// TwinCAT 3 PLC project HARTL_PowerLink_v2_03
// ProgramVersion: 3.1.4023.0
// libraries:
//   EfficientIO Communicator, * (EfficientIO)
//   EfficientIO ModbusTCP, * (EfficientIO)
//   Lynus Energy Basic, * (Lynus AG)
//   Lynus Persistent Data V1, * (Lynus AG)
//   Lynus Standards, * (Lynus AG)
//   Tc2_BABasic, * (Beckhoff Automation GmbH)
//   Tc2_ModbusSrv, * (Beckhoff Automation GmbH)
//   Tc2_Standard, * (Beckhoff Automation GmbH)
//   Tc2_System, * (Beckhoff Automation GmbH)
//   Tc2_Utilities, * (Beckhoff Automation GmbH)
//   Tc3_Module, * (Beckhoff Automation GmbH)
// project tree:
//   / FastTask.TcTTO, MiddleTask.TcTTO, SlowTask.TcTTO (not stored)
//   FBs/ FB_EM24_DIN.TcPOU (not stored), FB_Enphase.TcPOU, FB_Enphase_Helper.TcPOU (not stored), FB_ModBus_100Registers_FC3_inclID.TcPOU (not stored)
//   POUs/ prgBattery.TcPOU (not stored), prgCalc.TcPOU, prgComEffIO.TcPOU, prgEM.TcPOU, prgEMS.TcPOU, prgEnphase.TcPOU, prgPersistent.TcPOU (not stored), prgPV.TcPOU (not stored), prgCS.TcPOU, prgRWEffIO.TcPOU (not stored), prgSystemTime.TcPOU (not stored), prgVarEffIO.TcPOU (not stored)
// real-time tasks:
//   TASK FastTask: cycle T#5ms, priority 19, ADS port 350
//   TASK MiddleTask: cycle T#10ms, priority 20, ADS port 351
//   TASK SlowTask: cycle T#20ms, priority 21, ADS port 352
// I/O:
//   DEVICE Device 1 (Beckhoff CCAT)
//   DEVICE Device 2 (CX-BK)
//     Box 1 (CX-BK)
// variable links:
//   HARTL_PowerLink_v2_03/HARTL_PowerLink_v2_03 Instance <-> Device 2 (CX-BK)/Box 1 (CX-BK)
//     MiddleTask Inputs/prgEM.fbEM1.fbKL3403.byStateCH1 <-> Term 2 (KL3403)/Channel 1/State
//     MiddleTask Inputs/prgEM.fbEM1.fbKL3403.byStateCH2 <-> Term 2 (KL3403)/Channel 2/State
//     MiddleTask Inputs/prgEM.fbEM1.fbKL3403.byStateCH3 <-> Term 2 (KL3403)/Channel 3/State
//     MiddleTask Inputs/prgEM.fbEM2.fbKL3403.byStateCH1 <-> Term 3 (KL3403)/Channel 1/State
//     MiddleTask Inputs/prgEM.fbEM2.fbKL3403.byStateCH2 <-> Term 3 (KL3403)/Channel 2/State
//     MiddleTask Inputs/prgEM.fbEM2.fbKL3403.byStateCH3 <-> Term 3 (KL3403)/Channel 3/State
//     MiddleTask Inputs/prgEM.fbEM3.fbKL3403.byStateCH1 <-> Term 4 (KL3403)/Channel 1/State
//     MiddleTask Inputs/prgEM.fbEM3.fbKL3403.byStateCH2 <-> Term 4 (KL3403)/Channel 2/State
//     MiddleTask Inputs/prgEM.fbEM3.fbKL3403.byStateCH3 <-> Term 4 (KL3403)/Channel 3/State
//     MiddleTask Inputs/prgEM.fbEM4.fbKL3403.byStateCH1 <-> Term 5 (KL3403)/Channel 1/State
//     MiddleTask Inputs/prgEM.fbEM4.fbKL3403.byStateCH2 <-> Term 5 (KL3403)/Channel 2/State
//     MiddleTask Inputs/prgEM.fbEM4.fbKL3403.byStateCH3 <-> Term 5 (KL3403)/Channel 3/State
//     MiddleTask Inputs/prgEM.fbEM1.fbKL3403.iDataInCH1 <-> Term 2 (KL3403)/Channel 1/Data In
//     MiddleTask Inputs/prgEM.fbEM1.fbKL3403.iDataInCH2 <-> Term 2 (KL3403)/Channel 2/Data In
//     MiddleTask Inputs/prgEM.fbEM1.fbKL3403.iDataInCH3 <-> Term 2 (KL3403)/Channel 3/Data In
//     MiddleTask Inputs/prgEM.fbEM2.fbKL3403.iDataInCH1 <-> Term 3 (KL3403)/Channel 1/Data In
//     MiddleTask Inputs/prgEM.fbEM2.fbKL3403.iDataInCH2 <-> Term 3 (KL3403)/Channel 2/Data In
//     MiddleTask Inputs/prgEM.fbEM2.fbKL3403.iDataInCH3 <-> Term 3 (KL3403)/Channel 3/Data In
//     MiddleTask Inputs/prgEM.fbEM3.fbKL3403.iDataInCH1 <-> Term 4 (KL3403)/Channel 1/Data In
//     MiddleTask Inputs/prgEM.fbEM3.fbKL3403.iDataInCH2 <-> Term 4 (KL3403)/Channel 2/Data In
//     MiddleTask Inputs/prgEM.fbEM3.fbKL3403.iDataInCH3 <-> Term 4 (KL3403)/Channel 3/Data In
//     MiddleTask Inputs/prgEM.fbEM4.fbKL3403.iDataInCH1 <-> Term 5 (KL3403)/Channel 1/Data In
//     MiddleTask Inputs/prgEM.fbEM4.fbKL3403.iDataInCH2 <-> Term 5 (KL3403)/Channel 2/Data In
//     MiddleTask Inputs/prgEM.fbEM4.fbKL3403.iDataInCH3 <-> Term 5 (KL3403)/Channel 3/Data In
//     MiddleTask Inputs/prgEM.fbKBusState.uiKBusState_OUT <-> Inputs/State
//     MiddleTask Outputs/prgEM.fbEM1.fbKL3403.byCntrCH1 <-> Term 2 (KL3403)/Channel 1/Ctrl
//     MiddleTask Outputs/prgEM.fbEM1.fbKL3403.byCntrCH2 <-> Term 2 (KL3403)/Channel 2/Ctrl
//     MiddleTask Outputs/prgEM.fbEM1.fbKL3403.byCntrCH3 <-> Term 2 (KL3403)/Channel 3/Ctrl
//     MiddleTask Outputs/prgEM.fbEM2.fbKL3403.byCntrCH1 <-> Term 3 (KL3403)/Channel 1/Ctrl
//     MiddleTask Outputs/prgEM.fbEM2.fbKL3403.byCntrCH2 <-> Term 3 (KL3403)/Channel 2/Ctrl
//     MiddleTask Outputs/prgEM.fbEM2.fbKL3403.byCntrCH3 <-> Term 3 (KL3403)/Channel 3/Ctrl
//     MiddleTask Outputs/prgEM.fbEM3.fbKL3403.byCntrCH1 <-> Term 4 (KL3403)/Channel 1/Ctrl
//     MiddleTask Outputs/prgEM.fbEM3.fbKL3403.byCntrCH2 <-> Term 4 (KL3403)/Channel 2/Ctrl
//     MiddleTask Outputs/prgEM.fbEM3.fbKL3403.byCntrCH3 <-> Term 4 (KL3403)/Channel 3/Ctrl
//     MiddleTask Outputs/prgEM.fbEM4.fbKL3403.byCntrCH1 <-> Term 5 (KL3403)/Channel 1/Ctrl
//     MiddleTask Outputs/prgEM.fbEM4.fbKL3403.byCntrCH2 <-> Term 5 (KL3403)/Channel 2/Ctrl
//     MiddleTask Outputs/prgEM.fbEM4.fbKL3403.byCntrCH3 <-> Term 5 (KL3403)/Channel 3/Ctrl
//     MiddleTask Outputs/prgEMS.bQ1State <-> Term 6 (KL2012)/Channel 1/Output
//     MiddleTask Outputs/prgEMS.bQ2State <-> Term 6 (KL2012)/Channel 2/Output
//     MiddleTask Outputs/prgEMS.bQ3State <-> Term 7 (KL2012)/Channel 1/Output
//     MiddleTask Outputs/prgEMS.bQ4State <-> Term 7 (KL2012)/Channel 2/Output

CONFIGURATION HARTL_PowerLink_v2_03
    RESOURCE PLC ON TwinCAT3
        TASK FastTask(INTERVAL := T#5ms, PRIORITY := 19);
        TASK MiddleTask(INTERVAL := T#10ms, PRIORITY := 20);
        PROGRAM prgRWEffIO WITH FastTask : prgRWEffIO;
        PROGRAM prgVarEffIO WITH FastTask : prgVarEffIO;
        PROGRAM prgEM WITH MiddleTask : prgEM;
        PROGRAM prgEMS WITH MiddleTask : prgEMS;
        PROGRAM prgSystemTime WITH MiddleTask : prgSystemTime;
        PROGRAM prgCS WITH MiddleTask : prgCS;
        PROGRAM prgPersistent WITH MiddleTask : prgPersistent;
        PROGRAM prgCalc WITH MiddleTask : prgCalc;
    END_RESOURCE
END_CONFIGURATION

// ---- POUs/prgEM.TcPOU
PROGRAM prgEM
VAR
	fbKBusState		: FB_K_Bus_State;
	fbEM1			: FB_EM_Beckhoff_KL3403;
	fbEM1Counter	: FB_EnergyCounter;
	fbEM2			: FB_EM_Beckhoff_KL3403;
	fbEM2Counter	: FB_EnergyCounter;
	fbEM3			: FB_EM_Beckhoff_KL3403;
	fbEM3Counter	: FB_EnergyCounter;
	fbEM4			: FB_EM_Beckhoff_KL3403;
	fbEM4Counter	: FB_EnergyCounter;
	lrPowerEM1		: LREAL;						//{#lynus.ag#()}
	lrPowerEM2		: LREAL;						//{#lynus.ag#()}
	lrPowerEM3		: LREAL;						//{#lynus.ag#()}
	lrPowerEM4		: LREAL;						//{#lynus.ag#()}
	lr_InputVoltage_L1N		: LREAL;						//{#lynus.ag#()}
	lr_InputVoltage_L2N		: LREAL;						//{#lynus.ag#()}
	lr_InputVoltage_L3N		: LREAL;						//{#lynus.ag#()}
	lr_InputVoltage_L1L2	: LREAL;						//{#lynus.ag#()}
	lr_InputVoltage_L2L3	: LREAL;						//{#lynus.ag#()}
	lr_InputVoltage_L3L1	: LREAL;						//{#lynus.ag#()}
END_VAR
VAR PERSISTENT
	lrCounterEM1	: LREAL;						//{#lynus.ag#()}
	lrCounterEM2	: LREAL;						//{#lynus.ag#()}
	lrCounterEM3	: LREAL;						//{#lynus.ag#()}
	lrCounterEM4	: LREAL;						//{#lynus.ag#()}
END_VAR

fbKBusState(uiKBusState_OUT=> );

// Base Connection

fbEM1(
	bEnable:= TRUE, 
	bChannel1Invers:= FALSE,
	bChannel2Invers:= FALSE,
	bChannel3Invers:= FALSE,
	uiCurrentTransformerRatioL1:= 64, 
	uiCurrentTransformerRatioL2:= 64, 
	uiCurrentTransformerRatioL3:= 64, 
	uiKBusState_IN:= fbKBusState.uiKBusState_OUT, 
	stDataEMPower=> , 
	stDataEMCounter=> , 
	stDataEMPowerRealTime=> , 
	stDataEMCounterRealTime=> , 
	diNrOfEM_OUT=> );

lrPowerEM1 := fbEM1.stDataEMPower.lrPowerTotal;
lr_InputVoltage_L1N := fbEM1.stDataEMPower.lrVoltageL1N;
lr_InputVoltage_L2N := fbEM1.stDataEMPower.lrVoltageL2N;
lr_InputVoltage_L3N := fbEM1.stDataEMPower.lrVoltageL3N;
lr_InputVoltage_L1L2 := fbEM1.stDataEMPower.lrVoltageL1L2;
lr_InputVoltage_L2L3 := fbEM1.stDataEMPower.lrVoltageL2L3;
lr_InputVoltage_L3L1 := fbEM1.stDataEMPower.lrVoltageL3L1;

fbEM1Counter(
	byActiveTariff:= 1, 
	lrPowerInput:= lrPowerEM1, 
	lrTotalCounterEnergy_Consumption=> , 
	lrTotalCounterEnergy_Production=> , 
	lrCounterEnergyT1_Consumption=> , 
	lrCounterEnergyT2_Consumption=> , 
	lrCounterEnergyT1_Production=> , 
	lrCounterEnergyT2_Production=> );
	
IF fbEM1Counter.lrTotalCounterEnergy_Consumption > lrCounterEM1 THEN  	
	lrCounterEM1 := fbEM1Counter.lrTotalCounterEnergy_Consumption;
END_IF

// Output1, 3x400V 32A, CEE32

fbEM2(
	bEnable:= TRUE, 
	bChannel1Invers:= FALSE,
	bChannel2Invers:= FALSE,
	bChannel3Invers:= FALSE,
	uiCurrentTransformerRatioL1:= 35, 
	uiCurrentTransformerRatioL2:= 35, 
	uiCurrentTransformerRatioL3:= 35, 
	uiKBusState_IN:= fbKBusState.uiKBusState_OUT, 
	stDataEMPower=> , 
	stDataEMCounter=> , 
	stDataEMPowerRealTime=> , 
	stDataEMCounterRealTime=> , 
	diNrOfEM_OUT=> );

lrPowerEM2 := fbEM2.stDataEMPower.lrPowerTotal;	

fbEM2Counter(
	byActiveTariff:= 1, 
	lrPowerInput:= lrPowerEM2, 
	lrTotalCounterEnergy_Consumption=> , 
	lrTotalCounterEnergy_Production=> , 
	lrCounterEnergyT1_Consumption=> , 
	lrCounterEnergyT2_Consumption=> , 
	lrCounterEnergyT1_Production=> , 
	lrCounterEnergyT2_Production=> );
	
IF fbEM2Counter.lrTotalCounterEnergy_Consumption > lrCounterEM2 THEN  	
	lrCounterEM2 := fbEM2Counter.lrTotalCounterEnergy_Consumption;
END_IF


// Output2, 3x400V 32A, CEE32

fbEM3(
	bEnable:= TRUE, 
	bChannel1Invers:= FALSE,
	bChannel2Invers:= FALSE,
	bChannel3Invers:= FALSE,
	uiCurrentTransformerRatioL1:= 35, 
	uiCurrentTransformerRatioL2:= 35, 
	uiCurrentTransformerRatioL3:= 35, 
	uiKBusState_IN:= fbKBusState.uiKBusState_OUT, 
	stDataEMPower=> , 
	stDataEMCounter=> , 
	stDataEMPowerRealTime=> , 
	stDataEMCounterRealTime=> , 
	diNrOfEM_OUT=> );

lrPowerEM3 := fbEM3.stDataEMPower.lrPowerTotal;	

fbEM3Counter(
	byActiveTariff:= 1, 
	lrPowerInput:= lrPowerEM3, 
	lrTotalCounterEnergy_Consumption=> , 
	lrTotalCounterEnergy_Production=> , 
	lrCounterEnergyT1_Consumption=> , 
	lrCounterEnergyT2_Consumption=> , 
	lrCounterEnergyT1_Production=> , 
	lrCounterEnergyT2_Production=> );
	
IF fbEM3Counter.lrTotalCounterEnergy_Consumption > lrCounterEM3 THEN  	
	lrCounterEM3 := fbEM3Counter.lrTotalCounterEnergy_Consumption;
END_IF


// Output3, 3x400V 16A, CEE16

fbEM4(
	bEnable:= TRUE, 
	bChannel1Invers:= FALSE,
	bChannel2Invers:= FALSE,
	bChannel3Invers:= FALSE,
	uiCurrentTransformerRatioL1:= 35, 
	uiCurrentTransformerRatioL2:= 35, 
	uiCurrentTransformerRatioL3:= 35, 
	uiKBusState_IN:= fbKBusState.uiKBusState_OUT, 
	stDataEMPower=> , 
	stDataEMCounter=> , 
	stDataEMPowerRealTime=> , 
	stDataEMCounterRealTime=> , 
	diNrOfEM_OUT=> );

lrPowerEM4 := fbEM4.stDataEMPower.lrPowerTotal;	

fbEM4Counter(
	byActiveTariff:= 1, 
	lrPowerInput:= lrPowerEM4, 
	lrTotalCounterEnergy_Consumption=> , 
	lrTotalCounterEnergy_Production=> , 
	lrCounterEnergyT1_Consumption=> , 
	lrCounterEnergyT2_Consumption=> , 
	lrCounterEnergyT1_Production=> , 
	lrCounterEnergyT2_Production=> );
	
IF fbEM4Counter.lrTotalCounterEnergy_Consumption > lrCounterEM4 THEN  	
	lrCounterEM4 := fbEM4Counter.lrTotalCounterEnergy_Consumption;
END_IF

END_PROGRAM

// ---- POUs/prgEMS.TcPOU
PROGRAM prgEMS
VAR
	// Q1, 3x400V 32A, CEE32
	RS_Q1						: RS;
	bQ1On						: BOOL;						//{#lynus.ag#()}
	bQ1Off						: BOOL;						//{#lynus.ag#()}
	bQ1State	AT%Q*			: BOOL;						//{#lynus.ag#()}
	bQ1State_NOT				: BOOL;						//{#lynus.ag#()}
	// Q2, 3x400V 32A, CEE32
	RS_Q2						: RS;
	bQ2On						: BOOL;						//{#lynus.ag#()}
	bQ2Off						: BOOL;						//{#lynus.ag#()}
	bQ2State	AT%Q*			: BOOL;						//{#lynus.ag#()}
	bQ2State_NOT				: BOOL;						//{#lynus.ag#()}
	// Q3, 3x400V 16A, CEE16
	RS_Q3						: RS;	
	bQ3On						: BOOL;						//{#lynus.ag#()}
	bQ3Off						: BOOL;						//{#lynus.ag#()}
	bQ3State	AT%Q*			: BOOL;						//{#lynus.ag#()}
	bQ3State_NOT				: BOOL;						//{#lynus.ag#()}
	// Q4, 3x400V 16A, CEE16, EV Charging
	RS_Q4						: RS;
	bQ4On						: BOOL;						//{#lynus.ag#()}
	bQ4Off						: BOOL;						//{#lynus.ag#()}
	bQ4State	AT%Q*			: BOOL;						//{#lynus.ag#()}
	bQ4State_NOT				: BOOL;						//{#lynus.ag#()}
	
	// Automatic PV-Inverter Shutdown
	fbNFS_PV					: FB_WeeklyTimeSwitch;
	fbCalcSunriseSunset   		: FB_CalcSunriseSunset;
	todSunrise            		: TOD;
	todSunset             		: TOD;
END_VAR
VAR PERSISTENT
	bEnableNFS_PV				: BOOL;						//{#lynus.ag#()}
END_VAR

// To-Do:
// adopt Longitude and Latitude
// set bEdgeOn and bEdgeOff to correct Q Variables

// Output Controls
RS_Q1(SET:=bQ1Off , RESET1:=bQ1On , Q1=> bQ1State);
RS_Q2(SET:=bQ2Off , RESET1:=bQ2On , Q1=> bQ2State);
RS_Q3(SET:=bQ3Off , RESET1:=bQ3On , Q1=> bQ3State);
RS_Q4(SET:=bQ4Off , RESET1:=bQ4On , Q1=> bQ4State);
bQ1State_NOT := NOT bQ1State;
bQ2State_NOT := NOT bQ2State;
bQ3State_NOT := NOT bQ3State;
bQ4State_NOT := NOT bQ4State;

// fbQ1(bOn:=bQ1Off, bOff:=bQ1On, bLight=>bQ1State);
// fbQ2(bOn:=bQ2Off, bOff:=bQ2On, bLight=>bQ2State);
// fbQ3(bOn:=bQ3Off, bOff:=bQ3On, bLight=>bQ3State);
// fbQ4(bOn:=bQ4Off, bOff:=bQ4On, bLight=>bQ4State);

// Sunrise, Sunset calc
IF prgSystemTime.bSystemTimeValid THEN

	fbCalcSunriseSunset(
		fDegreeOfLongitude := 11.5820,   (* Longitude of Munich, Lochhausen *)
        fDegreeOfLatitude := 48.1351,   (* Latitude of Munich, Lochhausen *)
    	fReferenceMeridian := 15.0,  (* Central European Time *)
        dCurrentDate := DT_TO_DATE(prgSystemTime.dtSystemTime),
        todSunrise => todSunrise,
        todSunset => todSunset);
END_IF

// Automatic PV-Inverter Shutdown
IF prgSystemTime.bSystemTimeValid THEN
	fbNFS_PV(
		bEnable:=bEnableNFS_PV, 
		tCurrentDateTime:=prgSystemTime.dtSystemTime, 
		tSwitchOnTime:=todSunrise, 
		tSwitchOffTime:=todSunset, 
		bSunday:=TRUE, 
		bMonday:=TRUE, 
		bTuesday:=TRUE, 
		bWednesday:=TRUE, 
		bThursday:=TRUE, 
		bFriday:=TRUE, 
		bSaturday:=TRUE,
		bEdgeOn=> ,
		bEdgeOff=> );
END_IF

END_PROGRAM

// ---- POUs/prgCS.TcPOU
PROGRAM prgCS
VAR
	fbCS						: FB_EM24_DIN; 
	fbCSCounter					: FB_EnergyCounter;
	lrPowerCS					: LREAL;						//{#lynus.ag#()}
	// udintErrorWarningCS			: UDINT;
	FB_MB_Test :FB_ModBus_100Registers_FC3_inclID;
	
END_VAR
VAR PERSISTENT
	lrCounterCS					: LREAL;						//{#lynus.ag#()}
	lrCounterCSeIO				: LREAL;						//{#lynus.ag#()}
END_VAR

// To-Do:
// adopt FB Declaration, change to new FB for ENERGYMID
// adopt FB Definition, change to correct in/out Vars for ENERGYMID
// correct lrPowerCS definition
// correct lrCounterCS definition
// correct byErrorWarningCS definition
fbCS(
	m_Enable:= , 
	str_IPAdress:= '192.168.1.20', 
	real_RealPower_kW=> , 
	real_RealPowerL1_kW=> , 
	real_RealPowerL2_kW=> , 
	real_RealPowerL3_kW=> , 
	real_ReactivePower_kVAr=> , 
	real_ApparentPower_kVA=> , 
	real_Frequency_Hz=> , 
	real_VoltageL1N_V=> , 
	real_VoltageL2N_V=> , 
	real_VoltageL3N_V=> , 
	real_VoltageL1L2_V=> , 
	real_VoltageL2L3_V=> , 
	real_VoltageL3L1_V=> , 
	real_CurrentL1_A=> , 
	real_CurrentL2_A=> , 
	real_CurrentL3_A=> , 
	real_EnergyTotal_Import_kWh=> , 
	real_EnergyTotal_Export_kWh=> , 
	real_EnergyTotal_ExportT1_kWh=> , 
	real_EnergyTotal_ExportT2_kWh=> , 
	real_EnergyTotal_ExportT3_kWh=> , 
	real_EnergyTotal_ExportT4_kWh=> , 
	m_PollSuccessful=> , 
	udint_Error_ID=> );
(*fbCS(
	m_Enable:= , //TRUE, 
	str_IPAdress:= '192.168.1.20', 
	real_EnergyTotal_Wh => , 
	real_RealPower_W => ,
	udint_Error_ID =>);*)

lrPowerCS := fbCS.real_RealPower_kW;
// uErrorWarningCS := fbCS.udint_Error_ID;

// MID conform Counter, read from Energymeter
IF fbCS.real_EnergyTotal_Import_kWh > lrCounterCS THEN  	
	lrCounterCS := fbCS.real_EnergyTotal_Import_kWh;
END_IF

// internal Counter, for comparing purpose
fbCSCounter(
	byActiveTariff:= 1, 
	lrPowerInput:= lrPowerCS, 
	lrTotalCounterEnergy_Consumption=> , 
	lrTotalCounterEnergy_Production=> , 
	lrCounterEnergyT1_Consumption=> , 
	lrCounterEnergyT2_Consumption=> , 
	lrCounterEnergyT1_Production=> , 
	lrCounterEnergyT2_Production=> );
	
IF fbCSCounter.lrTotalCounterEnergy_Consumption > lrCounterCSeIO THEN  	
	lrCounterCSeIO := fbCSCounter.lrTotalCounterEnergy_Consumption;
END_IF

FB_MB_Test(
	m_Enable:= , 
	str_IPAdress:= '192.168.1.20', 
	w_Adress:= , 
	usint_Quantity:= , 
	usint_ID:= , 
	m_PollSuccessful=> , 
	w_Array_Received=> , 
	udint_Error_ID=> );

END_PROGRAM

// ---- POUs/prgCalc.TcPOU
PROGRAM prgCalc
VAR
	fbQ56Counter	: FB_EnergyCounter;
	lrPowerQ56		: LREAL;						//{#lynus.ag#()}
END_VAR
VAR PERSISTENT
	lrCounterQ56	: LREAL;						//{#lynus.ag#()}
	lrCO2Enphase	: LREAL;						//{#lynus.ag#()}
	lrCO2PV			: LREAL;						//{#lynus.ag#()}
END_VAR

// calc Output 5 & 6, 230V 16A, Schuko
// choose one of the two calc-options

// 1 -- if prgPV is in use
// lrPowerQ56 := (prgEM.lrPowerEM1 + prgBattery.lrPowerBatt + prgPV.lrPowerPV) - (prgEM.lrPowerEM2 + prgEM.lrPowerEM3 + prgEM.lrPowerEM4 + prgCS.lrPowerCS);
lrPowerQ56 := LIMIT(0,(prgEM.lrPowerEM1) - (prgEM.lrPowerEM2 + prgEM.lrPowerEM3 + prgEM.lrPowerEM4 + prgCS.lrPowerCS),10);

// 2 -- if prgEnphase is in use
// lrPowerQ56 := (prgEM.lrPowerEM1 + prgBattery.lrPowerBatt + prgEnphase.lrPowerPV) - (prgEM.lrPowerEM2 + prgEM.lrPowerEM3 + prgEM.lrPowerEM4 + prgCS.lrPowerCS);


// calc saved CO2
// lrCO2Enphase := prgEnphase.lrCounterPV * 0.428;
// lrCO2PV := prgPV.lrCounterPV * 0.428;

END_PROGRAM

// ---- FBs/FB_Enphase.TcPOU
FUNCTION_BLOCK FB_Enphase
VAR_INPUT
	bStart				: BOOL;
	tDelayRequest		: TIME := T#3S;		//Timer for delay before start with the next read or write Request
	sHostname			: STRING(255);		//Hostname or IP Adress from the Server
END_VAR

VAR_IN_OUT
END_VAR

VAR_OUTPUT
	bValidResult				: BOOL;															//Valid Result received from Server
    bBusy						: BOOL;															//Function is Busy
    bError						: BOOL;															//Error sucess
	bDone						: BOOL;															//True after the decoding from the received Json File
	bConnected					: BOOL;															//Connection to the Server
	lrpowerprod					: LREAL;														//Received Value
	lrpowercons					: LREAL;														//Received Value
	hrErrorCode       			: HRESULT;														//Error Result from Http Client
END_VAR

VAR
	fbClient					: FB_IotHttpClient;
	fbHttpGet					: FB_Enphase_Helper;
	timStartRequest				: TON;															//Timer to Start the Request
	FPStartRequest				: R_TRIG;														//Internal positive Edge
	FPDone						: R_TRIG;														//Internal positive Edge
	FNStart						: F_TRIG;														//Internal negative Edge
END_VAR

(*------------------------------------------------------------------------------------Configure HTTP Client------------------------------------------------------------------------------------------------------*)

fbClient.sHostName := sHostname;
fbClient.tConnectionTimeout := tDelayRequest;

IF NOT fbClient.bConfigured THEN 
	fbClient.nHostPort:= 80;
	fbClient.bKeepAlive := TRUE;
	fbClient.tConnectionTimeout := T#2S;
END_IF


//Timer to start the Request
FPStartRequest(CLK:= bStart, Q=> );
	timStartRequest(IN:= fbClient.bConfigured AND bStart AND NOT timStartRequest.Q, PT:= tDelayRequest, Q=> , ET=> );
		IF ((timStartRequest.Q AND NOT bBusy) OR (FPStartRequest.Q AND NOT bBusy AND fbClient.bConfigured)) THEN fbHttpGet.bSend := TRUE; END_IF

				
//Http Get Function
fbHttpGet(
	lrpowerprod => lrpowerprod, 
	lrpowercons => lrpowercons,
	bSend:= , 
	fbClient:= fbClient, 
	bBusy=> bBusy, 
	bError=> ,
	sContent=> );


fbHttpGet.bSend := FALSE;

FPDone(CLK:= bDone, Q=> );

(*
//Http Client
FNStart(CLK:= bStart, Q=> );
	IF FNStart.Q THEN fbClient.Disconnect(); END_IF
*)

fbClient.Execute();

//Error
IF fbHttpGet.bError OR fbClient.bError THEN bError := TRUE; ELSE bError := FALSE; END_IF	
	hrErrorCode := fbClient.hrErrorCode;

END_FUNCTION_BLOCK

// ---- POUs/prgComEffIO.TcPOU
PROGRAM prgComEffIO
VAR
	fbCom		: FB_MqttCommunicator_V2;
END_VAR

fbCom(
	bConnect:= TRUE, 
	strAuthkey := 'EIO08031879806',
	sUserName:= '21fb24f0-5311-4dec-a3c2-aacdaf7e170e', 
	sUserPassword:= '986af255-140d-48a9-82a9-cc9f22b85e6c', 
	eSavePositionCertificate:= eSavePositionOnPLC.ePostionHardDisk, 
	bConnected=> , 
	bError=> , 
	hrErrorCode=> , 
	eConnectionState=> , 
	eErrorMessage_Out=> );

END_PROGRAM

// ---- POUs/prgEnphase.TcPOU
PROGRAM prgEnphase
VAR
	fbEnphase					: FB_Enphase;
	fbPVCounter					: FB_EnergyCounter;
	fbGridCounter				: FB_EnergyCounter;
	lrPowerPV_W					: LREAL;
	lrPowerGrid_W				: LREAL;
	lrPowerPV					: LREAL;						//{#lynus.ag#()}
	lrPowerGrid					: LREAL;						//{#lynus.ag#()}
END_VAR

VAR PERSISTENT
	lrCounterPV					: LREAL;						//{#lynus.ag#()}
	lrCounterGrid				: LREAL;						//{#lynus.ag#()}
END_VAR

fbEnphase(
	bStart:= TRUE, 
	tDelayRequest:= T#3S, 
	sHostname:= '192.168.1.30', 
	bValidResult=> , 
	bBusy=> , 
	bError=> , 
	bDone=> , 
	hrErrorCode=> ,
	lrpowerprod => lrPowerPV_W,
	lrpowercons => lrPowerGrid_W );
	
// re-calc Power to kW
lrPowerPV := lrPowerPV_W / 1000;
lrPowerGrid := lrPowerGrid_W / 1000;

fbPVCounter(
	byActiveTariff:= 1, 
	lrPowerInput:= lrPowerPV, 
	lrTotalCounterEnergy_Consumption=> , 
	lrTotalCounterEnergy_Production=> , 
	lrCounterEnergyT1_Consumption=> , 
	lrCounterEnergyT2_Consumption=> , 
	lrCounterEnergyT1_Production=> , 
	lrCounterEnergyT2_Production=> );
	
IF fbPVCounter.lrTotalCounterEnergy_Consumption > lrCounterPV THEN  	
	lrCounterPV := fbPVCounter.lrTotalCounterEnergy_Consumption;
END_IF

fbGridCounter(
	byActiveTariff:= 1, 
	lrPowerInput:= lrPowerGrid, 
	lrTotalCounterEnergy_Consumption=> , 
	lrTotalCounterEnergy_Production=> , 
	lrCounterEnergyT1_Consumption=> , 
	lrCounterEnergyT2_Consumption=> , 
	lrCounterEnergyT1_Production=> , 
	lrCounterEnergyT2_Production=> );
	
IF fbGridCounter.lrTotalCounterEnergy_Consumption > lrCounterGrid THEN  	
	lrCounterGrid := fbGridCounter.lrTotalCounterEnergy_Consumption;
END_IF

END_PROGRAM
